// TwinCAT 3 PLC project DynamicDuos
// ProgramVersion: 3.1.4024.0
// libraries:
//   Tc2_Standard, * (Beckhoff Automation GmbH)
//   Tc2_System, * (Beckhoff Automation GmbH)
//   Tc2_Utilities, * (Beckhoff Automation GmbH)
//   Tc3_Module, * (Beckhoff Automation GmbH)
//   Haptix-Beckhoff,newest,HaptiX Lab
// project tree:
//   DUTs/ ActiveWindowStateType.TcDUT, CalibStateType.TcDUT, MainStateType.TcDUT, MasterStateType.TcDUT, ST_CalibLogChunk.TcDUT, ST_CalibrationSettings.TcDUT, ST_CalibTrialStep.TcDUT, ST_LoadExperimentSetting.TcDUT, ST_MainTrialStep.TcDUT
//   GVLs/ GVL.TcGVL
//   / PlcTask.TcTTO
//   POUs/ CalibrationBlock.TcPOU, CalibrationBlockLogger.TcPOU, CalibrationBlock_DOCILE.TcPOU, MAIN.TcPOU, MainExperimentBlock.TcPOU, MainExperimentBlockLogger.TcPOU, MAIN_DOCILE.TcPOU, TEST.TcPOU, WaitingMonitorBlock.TcPOU, MetadataBlock.TcPOU, MotorTorqueToCommandV.TcPOU
// real-time tasks:
//   TASK PlcTask: cycle T#100us, priority 4, ADS port 350
// I/O:
//   DEVICE Device 2 (EtherCAT), AmsNetId 141.212.76.55.3.1
//     Term 1 (EK1100) [EK1100 EtherCAT Coupler (2A E-Bus)]
//       Term 2 (EL4038) [EL4038 8Ch. Ana. Output +/-10V, 12bit]
//       Term 3 (EL3174) [EL3174 4Ch. Ana. Input +/-10V Diff., +/-20mA SingleEnded, 16 Bit]
//       Term 4 (EL5122) [EL5122 2Ch. Inc. Encoder 5V (2xAB TTL)]
//       Term 5 (EL9011) [EL9011 End Terminal]
// variable links:
//   DynamicDuos/DynamicDuos Instance <-> Device 2 (EtherCAT)/Term 1 (EK1100)/Term 2 (EL4038)
//     PlcTask Outputs/MAIN_DOCILE.fbMotor1.nNegAnalogOutput <-> AO Outputs Channel 2/Analog output
//     PlcTask Outputs/MAIN_DOCILE.fbMotor1.nPosAnalogOutput <-> AO Outputs Channel 1/Analog output
//     PlcTask Outputs/MAIN_DOCILE.fbMotor1.nZeroRefAnalogOutput <-> AO Outputs Channel 3/Analog output
//   DynamicDuos/DynamicDuos Instance <-> Device 2 (EtherCAT)/Term 1 (EK1100)/Term 3 (EL3174)
//     PlcTask Inputs/MAIN_DOCILE.fbLoadCell.nAnalogReading <-> AI Standard Channel 1/Value
//   DynamicDuos/DynamicDuos Instance <-> Device 2 (EtherCAT)/Term 1 (EK1100)/Term 4 (EL5122)
//     PlcTask Inputs/GVL.ENCODER_1_A_STATUS <-> ENC Status Channel 1/Status of input A
//     PlcTask Inputs/GVL.ENCODER_1_B_STATUS <-> ENC Status Channel 1/Status of input B
//     PlcTask Inputs/MAIN_DOCILE.fbEncoder1.QE_CHANNEL_COUNTS <-> ENC Status Channel 1/Counter value

CONFIGURATION DynamicDuos
    RESOURCE PLC ON TwinCAT3
        TASK PlcTask(INTERVAL := T#100us, PRIORITY := 4);
        PROGRAM MAIN_DOCILE WITH PlcTask : MAIN_DOCILE;
    END_RESOURCE
END_CONFIGURATION

// ---- DUTs/ActiveWindowStateType.TcDUT
{attribute 'qualified_only'}
{attribute 'strict'}
TYPE ActiveWindowStateType :
(
	EXPERIMENT_WINDOW := 0,
	CALIBRATION_WINDOW := 1, 
	PARTICIPANT_WINDOW := 2, 
	TRACKING_WINDOW := 3
) SINT := EXPERIMENT_WINDOW;
END_TYPE

// ---- DUTs/CalibStateType.TcDUT
{attribute 'qualified_only'}
{attribute 'strict'}
TYPE CalibStateType :
(
	PRE_LAUNCH := 0, // When the user is inputting settings. 
	TEST_SETUP := 1, // When the automation is getting the test ready
	TEST_ACTIVE := 2, // When the test is actively running. 
	TEST_FINISHED := 3, // When all calibration rounds have been completed. 
	ABORT := -1 // When the user has interrupted a test. 
	
);
END_TYPE

// ---- DUTs/MainStateType.TcDUT
{attribute 'qualified_only'}
{attribute 'strict'}
{attribute 'to_string'}
TYPE MainStateType :
(
	PRE_LAUNCH := 0, // When the user is inputting settings. 
	TEST_SETUP := 1, // When the automation is getting the test ready
	TEST_ACTIVE := 2, // When the test is actively running. 
	TEST_FINISHED := 3, // When all calibration rounds have been completed. 
	PROCESSING_LOG := 4, // When the log is saving.
	WAITING_FOR_RELEASE := 5, 
	ABORT := -1 // When the user has interrupted a test. 
);
END_TYPE

// ---- DUTs/MasterStateType.TcDUT
{attribute 'qualified_only'}
{attribute 'strict'}
{attribute 'to_string'}
TYPE MasterStateType :
(
	WAITING := 0, 
	CALIBRATION := 1, 
	ACTIVE := 2,
	TRACKING := 3, 
	ERROR := -1
)SINT := WAITING;
END_TYPE

// ---- DUTs/ST_CalibLogChunk.TcDUT
TYPE ST_CalibLogChunk :
STRUCT
	nChunkSizeBytes : DINT; 
	nChunkIndex : DINT; 
	nLastPointIndex : DINT := -1; // This will be positive if the last data point in an entire log lies within this chunk. The index will be the index of the last data point. 
	aChunk : ARRAY[0..GVL.MAX_CHUNK_SIZE] OF ST_CalibTrialStep;
END_STRUCT
END_TYPE

// ---- DUTs/ST_CalibrationSettings.TcDUT
TYPE ST_CalibrationSettings :
STRUCT
	bTestTypeHuman : BOOL; 
	nNumTrials : UINT;
	bTogglePulseWithGrip : BOOL;  
	bUseManualPulseTimer : BOOL; 
	bUseConstantGripTrigger : BOOL; 
	bUseConstantPulseTorque : BOOL; 
	rConstantPulseTorqueVal : REAL; 
	aGripSchedule : ARRAY[1..100] OF REAL; // There is never going to be 100, just some upper bound.
END_STRUCT
END_TYPE

// ---- DUTs/ST_CalibTrialStep.TcDUT
TYPE ST_CalibTrialStep : // Defines the configuration and data for a calibration trial at a given point in time. 
STRUCT
	nTimestepLow : UDINT;
	nTimeStepHigh : UDINT; 
	rEncoderDegrees : REAL; 
	rEncoderRadians : REAL; 
	rCommandVoltage : REAL; 
	rCommandTorque : REAL; 
	rAppliedTorque : REAL; 
	rVirtualSpringTorque : REAL; 
	rGripForce : REAL; 
	rCurrentGripThreshold : REAL; 
	sSequenceStateString : T_MaxString;  // String of the state
	nCurrentTestIndex : INT;
	nTestIsLive : INT; 
END_STRUCT
END_TYPE

// ---- DUTs/ST_LoadExperimentSetting.TcDUT
TYPE ST_LoadExperimentSetting :
STRUCT
	Weight : INT; 
	Test_Finished : BOOL; 
END_STRUCT
END_TYPE

// ---- DUTs/ST_MainTrialStep.TcDUT
TYPE ST_MainTrialStep :
STRUCT
	nTimestepLow : UDINT; 
	nTimestepHigh : UDINT; 
	rEncoderDegrees : REAL; 
	rEncoderRadians : REAL; 
	rCommandVoltage : REAL; 
	rCommandTorque : REAL; 
	rWallTorque : REAL; 
	rGripForce : REAL; 
	sSequenceStateString : T_MaxString; 
	nCurrentTestIndex : INT; 
	nTestIsLive : INT; 
END_STRUCT
END_TYPE

// ---- GVLs/GVL.TcGVL
{attribute 'qualified_only'}
VAR_GLOBAL

	ENCODER_1_DEGREES : REAL; 
	ENCODER_1_COUNTER_VALUE : LINT; 
	MOTOR_1_APPLIED_VOLTAGE : REAL; 
	ENCODER_1_A_STATUS AT %I* : BOOL; 
	ENCODER_1_B_STATUS AT %I* : BOOL;
	LOAD_CELL_NEWTONS : REAL; 
	MAIN_SYSTEM_TIME : UDINT; 
	CALIB_SYSTEM_TIME : UDINT; 
	
END_VAR

VAR_GLOBAL CONSTANT
	// Max amount of data entries we can 
	// send over the wire at once. 
	MAX_CHUNK_SIZE : DINT := 100; 
END_VAR

// ---- POUs/MAIN_DOCILE.TcPOU
PROGRAM MAIN_DOCILE
VAR
	
	// Variables for logging
	nEncoderCounts : LINT; 
	rEncoderDegrees : REAL;
	rEncoderLastDegrees : REAL; 
	rEncoderRadians : REAL; 
	rEncoderLastRadians : REAL; 
	rEncoderRadiansBuffer : ARRAY[1..FILTER_WINDOW] OF REAL; 
	rEncoderRadiansSum : REAL; 
	rEncoderRadiansFiltered : REAL; 
	nFilterBufferCount : INT := 0; 
	rGripForce : REAL; 
	
	// Sensors instantiation 
	fbEncoder1 : FB_QuadratureEncoder;
	fbLoadCell : FB_AnalogLoadCellInput;
	fbMotor1 : FB_AnalogMotorDriver;	

	
	// Helpers
	i : INT := 0;
	j : INT := 0;
	bIsFirstReset : BOOL := TRUE; 
	bEncoderReset : BOOL := FALSE; 
	fbSystemTime : GETSYSTEMTIME;
	
	stMasterState : MasterStateType := MasterStateType.WAITING; 
	
	
	// Child function block 
	{attribute 'OPC.UA.DA':='1'}
	fbCalibrationBlock : CalibrationBlock_DOCILE; 
	
	testCalibrationSettings : ST_CalibrationSettings; 

END_VAR
VAR CONSTANT
	// Constants for digital filtering 
	FILTER_WINDOW : INT := 11; 
END_VAR

// ===================================================== COMPLETE ALL SENSOR READINGS ========================================================
IF bIsFirstReset OR bEncoderReset THEN 
	fbEncoder1.Reset();
	bIsFirstReset := FALSE;
	bEncoderReset := FALSE; 
END_IF

// Encoders 
fbEncoder1(); 
nEncoderCounts := fbEncoder1.nNetCounts; 
rEncoderDegrees := fbEncoder1.rDegrees; 
rEncoderLastDegrees := fbEncoder1.rLastDegrees; 
rEncoderRadians := fbEncoder1.rRadians; 
rEncoderLastRadians := fbEncoder1.rLastRadians;

// Update digital filter. 
IF nFilterBufferCount < FILTER_WINDOW THEN 
	nFilterBufferCount := nFilterBufferCount + 1; 
END_IF

// Shift the buffer and add the new reading 
FOR i := FILTER_WINDOW TO 2 BY -1 DO
	rEncoderRadiansBuffer[i] := rEncoderRadiansBuffer[i-1]; 
END_FOR
rEncoderRadiansBuffer[1] := rEncoderRadians;

// Compute the moving average only if the buffer is full
j := MIN(nFilterBufferCount, FILTER_WINDOW); 
rEncoderRadiansSum := 0.0; 
FOR i:= 1 TO j DO
	rEncoderRadiansSum := rEncoderRadiansSum + rEncoderRadiansBuffer[i];
END_FOR
rEncoderRadiansFiltered := rEncoderRadiansSum / j; 

// Load cell   
fbLoadCell(); 
rGripForce := fbLoadCell.rCalibratedOutput; 
// ================================================ END SENSOR READINGS ==================================================

IF stMasterState = MasterStateType.CALIBRATION THEN 
	fbCalibrationBlock(
		rEncoderRadians := rEncoderRadians,
		rEncoderRadiansFiltered := rEncoderRadiansFiltered,
		rEncoderLastRadians := rEncoderLastRadians, 
		rGripForce := rGripForce,
		fbMotorReference := fbMotor1
	);
END_IF



// ================================================= UPDATE THE GVL ======================================================
GVL.ENCODER_1_DEGREES := fbEncoder1.rDegrees; 
GVL.LOAD_CELL_NEWTONS := rGripForce; 
fbSystemTime(timeLoDW => GVL.MAIN_SYSTEM_TIME);

END_PROGRAM

// ---- POUs/CalibrationBlock_DOCILE.TcPOU
FUNCTION_BLOCK CalibrationBlock_DOCILE
VAR_INPUT
	rEncoderRadians : REAL ;
	rEncoderRadiansFiltered : REAL; 
	rEncoderLastRadians : REAL;
	rGripForce : REAL; 
	fbMotorReference : REFERENCE TO FB_AnalogMotorDriver; 
END_VAR
VAR_OUTPUT
	rCommandVoltage : REAL;
	rVirtualSpringTorque : REAL;
	rAppliedTorque : REAL; 
	rCommandTorque : REAL; 
	rError : REAL;
	rLastError : REAL := 0;
	rProportional : REAL;
	rIntegral : REAL := 0;
	rDerivative : REAL; 
	bPIDStale : BOOL := TRUE; 
	rControlOutput : REAL;
	Kp : REAL := 0.3;
	Ki : REAL := 0.03;
	Kd : REAL := 0.05; 
	d_time : REAL := 0.0001; 
END_VAR
VAR
	z : INT := 0; 
	
	// State machine members for executing the test
	eSequenceState : CalibStateType := CalibStateType.PRE_LAUNCH; 
	eNextSequenceState : CalibStateType := CalibStateType.PRE_LAUNCH; 
	eSetupSubState : (HOMING, WAITING); 
	stCalibStepState : ST_CalibTrialStep; 
	stCalibrationSettings : ST_CalibrationSettings;
	
	// Virtual timers for accessing the test
	fbTonTest : TON := (PT := T#1000MS); // Timer for the entire test
	fbTonPulse : TON := (PT := T#200MS); // Timer for the duration of the pulse
	fbTonHoming : TON := (PT := T#500MS); // Time to give state machine to home
	bMotorLimitHit : BOOL := FALSE; 
	bWheelIsIdle : BOOL; 
	bTestIsLive : BOOL := FALSE; 
	bTestIsLiveTrigger : BOOL := FALSE; 
	rStartGripThreshold : REAL := 1.5;
	nCurrentTestIndex : INT := 0; 
	bLaunchTestSequence: BOOL;
	rCurrentGripThreshold : REAL := 100; // High number for init just so it can't go off by itself
	nCurrentLaunchIndex: INT := 0; 
	bLogHasBeenAcknowledged : BOOL := FALSE; 
	
	// Helper functions
	fbSystemTime : GETSYSTEMTIME; 
	nLastTimeStep : UDINT; 
	fbLogger : CalibrationBlockLogger; 
END_VAR

// Update the timers
fbTonTest(IN := bTestIsLive); 
fbTonPulse(IN := bTestIsLive);

CASE eSequenceState OF 
	
	// The user is currently setting prelaunch settings. 
	CalibStateType.PRE_LAUNCH: 
	
		// Make sure all variables are zerod 
		bTestIsLive := FALSE;
		rCommandVoltage := 0; 
		rVirtualSpringTorque := 0; 
		rAppliedTorque := 0; 
		rCommandTorque := 0; 
		fbMotorReference(rCommandVoltage := rCommandVoltage); 
	
		IF bLaunchTestSequence THEN // This would be set by the "LaunchTestSequence" method.
			eNextSequenceState := CalibStateType.TEST_SETUP; 
			
			// Also set the first test index
			nCurrentTestIndex := 1;  
			bLaunchTestSequence := FALSE; 
		ELSE
			eNextSequenceState := CalibStateType.PRE_LAUNCH; 
		END_IF
		
	// We are getting the test readt 
	CalibStateType.TEST_SETUP: 
	
		CASE eSetupSubState OF 
			HOMING: 
			
				bMotorLimitHit := FALSE; 
				
				// In this state, we need to recenter the motor back to the 0 point 
				// afterwards, we need to wait for the trigger signal 
				rError := 0 - rEncoderRadiansFiltered; 
				rProportional := Kp * rError; 
				rIntegral := rIntegral + (rError * d_time); 
				rDerivative := (rError - rLastError) / d_time; 
				rLastError := rError; 
				
				// On the first step, if the PID is stale, just use proportional 
				IF bPIDStale THEN 
					rAppliedTorque := rProportional; 
					rIntegral := 0; 
					bPIDStale := FALSE; 
				ELSE
					rAppliedTorque := rProportional + (Ki * rIntegral) + (Kd * rDerivative); 
				END_IF
				rVirtualSpringTorque := 0; 
				rCommandTorque := rAppliedTorque + rVirtualSpringTorque; 
				rCommandVoltage := MotorTorqueToCommandV(rCommandTorque := rCommandTorque); 
				fbMotorReference(rCommandVoltage := rCommandVoltage); 
				
				// Check to see if the wheel has been idle for ong enough 
				bWheelIsIdle := rGripForce < rStartGripThreshold AND ABS(rEncoderRadians) < 0.08;
				fbTonHoming(IN := bWheelIsIdle); 
				
				IF fbTonHoming.Q THEN 
					eSetupSubState := WAITING; 
				END_IF
				
			WAITING: 
				
				// Then we need to check if the test launch conditions are met 
				// We need to figure out the type of trigger being used
				IF bTestIsLiveTrigger AND NOT stCalibrationSettings.bTogglePulseWithGrip THEN
					bTestIsLive := TRUE; 
					bTestIsLiveTrigger := FALSE; 
				END_IF
				
				// If it's not the above, then we are toggling pulse with grip 
				IF  stCalibrationSettings.bTogglePulseWithGrip THEN 
					IF stCalibrationSettings.bUseConstantGripTrigger THEN 
						rCurrentGripThreshold := stCalibrationSettings.aGripSchedule[1]; 
					ELSE
						rCurrentGripThreshold := stCalibrationSettings.aGripSchedule[nCurrentTestIndex];
					END_IF 
					
					// Once we've set the value, we can compare to see if we've reached it
					IF rGripForce > rCurrentGripThreshold THEN 
						bTestIsLive := TRUE; 
					END_IF
					
				END_IF
				
				IF bTestIsLive THEN 
					eNextSequenceState := CalibStateType.TEST_ACTIVE; 
					bWheelIsIdle := FALSE; 
					fbTonHoming(IN := bWheelIsIdle); 
					eSetupSubState := HOMING; 
					bPIDStale := TRUE; 
				ELSE
					eNextSequenceState := CalibStateType.TEST_SETUP;
					// We need to let go of the motor
					rVirtualSpringTorque := 0; 
					rAppliedTorque := 0; 
					rCommandTorque := 0; 
					rCommandVoltage := 0;
					fbMotorReference(rCommandVoltage := rCommandVoltage); 
				END_IF
				
				
		END_CASE
		
		
	/// Then we handle the logic for actually completing the test 
	CalibStateType.TEST_ACTIVE: 
	
			// Timer is set based on the bTestIsLive variable. 
			IF NOT fbTonPulse.Q THEN 
			
				// We want to split motor action between motor test and human test mode. 
				// In motor test mode, we add a virtual spring so the motor doesn't slam into the bale
				IF NOT stCalibrationSettings.bTestTypeHuman THEN
					
					rAppliedTorque := stCalibrationSettings.rConstantPulseTorqueVal; 
					rVirtualSpringTorque := -1 * 0.35 * rEncoderRadians; 
				ELSE
					
					IF NOT stCalibrationSettings.bUseConstantPulseTorque THEN 
						rAppliedTorque := 0.4 + 0.02 * rCurrentGripThreshold; 
					ELSE
						rAppliedTorque := stCalibrationSettings.rConstantPulseTorqueVal; 
					END_IF 
					rVirtualSpringTorque := 0; 
			
				END_IF
				
				rCommandTorque := rAppliedTorque + rVirtualSpringTorque; 
				rCommandVoltage := MotorTorqueToCommandV(rCommandTorque := rCommandTorque); 
			ELSE
				
				IF NOT stCalibrationSettings.bTestTypeHuman THEN 
					rAppliedTorque := 0; 
					rVirtualSpringTorque := -1 * 0.35 * rEncoderRadians; 
				ELSE
					rAppliedTorque := 0; 
					rVirtualSpringTorque := 0; 
				END_IF
				
				rCommandTorque := rAppliedTorque + rVirtualSpringTorque; 
				rCommandVoltage := MotorTorqueToCommandV(rCommandTorque := rCommandTorque); 
			END_IF
			
			fbMotorReference(rCommandVoltage := rCommandVoltage); 
			
			// Now we check the test timer
			IF fbTonTest.Q THEN
				bTestIsLive := FALSE;
				IF nCurrentTestIndex < UINT_TO_INT(stCalibrationSettings.nNumTrials) THEN 
					nCurrentTestIndex := nCurrentTestIndex + 1; 
					eNextSequenceState := CalibStateType.TEST_SETUP; 
				ELSE
					eNextSequenceState := CalibStateType.TEST_FINISHED;
				END_IF
			END_IF
	
	CalibStateType.TEST_FINISHED: 
		// Do some logging 
		IF NOT bLogHasBeenAcknowledged THEN 
			eNextSequenceState := CalibStateType.TEST_FINISHED; 
		END_IF
		eNextSequenceState := CalibStateType.PROCESSING_LOG;
		
	CalibStateType.PROCESSING_LOG: 
		// Wait to see if logging finished
		nCurrentTestIndex := 0; 
		nCurrentLaunchIndex := nCurrentLaunchIndex + 1; 
		eNextSequenceState := CalibStateType.PRE_LAUNCH; 
END_CASE


// At the end of the main loop is when we actually do the logging 
nLastTimeStep := stCalibStepState.nTimestepLow; 
fbSystemTime(timeLoDW => stCalibStepState.nTimestepLow, timeHiDW => stCalibStepState.nTimeStepHigh); 
stCalibStepState.rEncoderDegrees := RAD_TO_DEG(rEncoderRadians); 
stCalibStepState.rEncoderRadians := rEncoderRadians; 
stCalibStepState.rCommandVoltage := rCommandVoltage; 
stCalibStepState.rCommandTorque := rCommandTorque; 
stCalibStepState.rAppliedTorque := rAppliedTorque; 
stCalibStepState.rVirtualSpringTorque := rVirtualSpringTorque; 
stCalibStepState.rGripForce := rGripForce; 
stCalibStepState.rCurrentGripThreshold := rCurrentGripThreshold; 
stCalibStepState.sSequenceStateString := TO_STRING(eSequenceState); 
stCalibStepState.nCurrentTestIndex := nCurrentTestIndex; 
stCalibStepState.nTestIsLive := BOOL_TO_INT(bTestIsLive); 

IF eSequenceState = CalibStateType.TEST_ACTIVE THEN
	fbLogger.addStep(stNewStep := stCalibStepState);
END_IF

// Update sequence state for next iteration 
eSequenceState := eNextSequenceState;

END_FUNCTION_BLOCK

// ---- POUs/CalibrationBlockLogger.TcPOU
FUNCTION_BLOCK CalibrationBlockLogger
VAR_INPUT
	sFileName : STRING; 
END_VAR
VAR_OUTPUT
	bBusy : BOOL := FALSE; 
	bError : BOOL := FALSE; 
END_VAR
VAR CONSTANT
	nMaxBufferSize : UDINT := 2000000;
END_VAR
VAR
	cDefaultHeader : T_MaxString := 'TimeLow,TimeHigh,EncoderDegrees,EncoderRadians,CommandVoltage,CommandTorque,AppliedTorque,VSTorque,GripForce,GripThreshold,SequenceState,CurrentTestIndex,TestIsLive $n'; 
	sDefaultDirectory : T_MaxString := 'C:\Users\njanne\Documents\DDTestLogs\calibration\'; 
	bWriteToDisk : BOOL := FALSE; 
	eFileWriteState : (IDLE, OPEN, WRITE, CLOSE, ERROR); 
	nFileWriteSubstep : INT := 0; 
	fbFileOpen : FB_FileOpen; 
	fbFilePuts : FB_FilePuts; 
	fbFileClose : FB_FileClose; 
	fbFormatString : FB_FormatString2; 
	nFileHandle : UINT; 
	bHeaderWriteComplete : BOOL := FALSE; 
	nWriteIndex : UDINT := 0; 
	sWritePercentFormat : T_MaxString := '%.2f %%'; 
	rWritePercent : REAL; 
	sWritePercentString : T_MaxString; 
	
	// For formatting data into a string. 
	sDataFormatStr1 : STRING := '%d,%d,%f,%f,%f,%f,%f,'; 
	sDataFormatStr2 : STRING := '%f,%f,%f,%s,%d,%d $n';
	sTempString : STRING(600); 
	sOutputString : STRING(600); 
	
	aTrialDataBuffer : ARRAY[0..nMaxBufferSize] OF ST_CalibTrialStep; 
	nStepsSoFar : UDINT := 0; // Current number of steps in the database. 
	
END_VAR

IF bWriteToDisk THEN

	// If it's time to write to disk, we need to empty the buffer.
	CASE eFileWriteState OF 
		
		IDLE: 
			// Get everything ready. 
			nFileHandle := 0; 
			bBusy := TRUE; 
			eFileWriteState := OPEN;
			nFileWriteSubstep := 0;  
	
		OPEN:
			CASE nFileWriteSubstep OF
				0:  
					// Opens a file for writing at the end of the file (append). 
					// If the file does not exist, a new file is created. 
					fbFileOpen(spathName := CONCAT(sDefaultDirectory, sFilename), bExecute := FALSE); 
					fbFileOpen(
						bExecute 		:= TRUE, 
						sNetID			:= '',
						sPathName 		:= CONCAT(sDefaultDirectory, sFilename), 
						nMode 			:= FOPEN_MODEAPPEND OR FOPEN_MODETEXT); 
		
					nFileWriteSubstep := nFileWriteSubstep + 1; // Advance to waiting state. 
	
				1: 
					fbFileOpen(bExecute := FALSE); 
					IF NOT fbFileOpen.bBusy THEN 
						IF fbFileOpen.bError THEN 
							eFileWriteState := ERROR; 
							nFileWriteSubstep := 0; 
						ELSE
							nFileHandle := fbFileOpen.hFile; 
							eFileWriteState := WRITE; 
							nFileWriteSubstep := 0; 
						END_IF
					END_IF
				END_CASE

		WRITE: 
			CASE nFileWriteSubstep OF 
				0 :
					fbFilePuts(bExecute := FALSE); 
					
					// Check if we still need to write the header. 
					IF NOT bHeaderWriteComplete THEN
						fbFilePuts(
							bExecute		:= TRUE, 
							sNetId			:= '', 
							hFile			:= nFileHandle, 
							sLine			:= cDefaultHeader);
						bHeaderWriteComplete := TRUE; 
					ELSE
						// If the header is already written, then we're going for data. 
						// We need to first format the string. 		
						fbFormatString(
							pFormatString := ADR(sDataFormatStr1), 
							arg1 := F_UDINT(aTrialDataBuffer[nWriteIndex].nTimestepLow), 
							arg2 := F_UDINT(aTrialDataBuffer[nWriteIndex].nTimeStepHigh),
							arg3 := F_REAL(aTrialDataBuffer[nWriteIndex].rEncoderDegrees), 
							arg4 := F_REAL(aTrialDataBuffer[nWriteIndex].rEncoderRadians), 
							arg5 := F_REAL(aTrialDataBuffer[nWriteIndex].rCommandVoltage), 
							arg6 := F_REAL(aTrialDataBuffer[nWriteIndex].rCommandTorque), 
							arg7 := F_REAL(aTrialDataBuffer[nWriteIndex].rAppliedTorque), 
							pDstString := ADR(sOutputString), 
							nDstSize := SIZEOF(sOutputString)); 
					
						fbFormatString(
							pFormatString := ADR(sDataFormatStr2), 
							arg1 := F_REAL(aTrialDataBuffer[nWriteIndex].rVirtualSpringTorque), 
							arg2 := F_REAL(aTrialDataBuffer[nWriteIndex].rGripForce), 
							arg3 := F_REAL(aTrialDataBuffer[nWriteIndex].rCurrentGripThreshold), 
							arg4 := F_STRING(aTrialDataBuffer[nWriteIndex].sSequenceStateString), 
							arg5 := F_INT(aTrialDataBuffer[nWriteIndex].nCurrentTestIndex), 
							arg6 := F_INT(aTrialDataBuffer[nWriteIndex].nTestIsLive), 
							pDstString := ADR(sTempString), 
							nDstSize := SIZEOF(sTempString)); 
							
						CONCAT2(
							pSrcString1 := ADR(sOutputString), 
							pSrcString2 := ADR(sTempString), 
							pDstString := ADR(sOutputString), 
							nDstSize := SIZEOF(sOutputString)); 
						
						fbFilePuts(
							bExecute		:= TRUE, 
							sNetId			:= '', 
							hFile			:= nFileHandle, 
							sLine			:= sOutputString); 
							
						nWriteIndex := nWriteIndex + 1; 
						// Update write progress 
						rWritePercent := UDINT_TO_REAL(nWriteIndex) / UDINT_TO_REAL(nStepsSoFar) * 100; 
						fbFormatString(
							pFormatString := ADR(sWritePercentFormat),
							arg1 := F_REAL(rWritePercent),
							pDstString := ADR(sWritePercentString), 
							nDstSize := SIZEOF(sWritePercentString)); 
				
					END_IF
					
					nFileWriteSubstep := nFileWriteSubstep + 1; // Advance to waiting state. 
					
				1 : 
					fbFilePuts(bExecute := FALSE); 
					IF NOT fbFilePuts.bBusy THEN
						IF fbFilePuts.bError THEN 
							eFileWriteState := ERROR; 
							nFileWriteSubstep := 0; 
						ELSE
							// Check if we have more things to write to the CSV still
							IF nWriteIndex = nStepsSoFar THEN
								eFileWriteState := CLOSE; 
							ELSE
								eFileWriteState := WRITE;
							END_IF 
						END_IF
						nFileWriteSubstep := 0; 
					END_IF
					
					
			END_CASE
		
		CLOSE: 
			CASE nFileWriteSubstep OF
				0: 
					fbFileClose(bExecute := FALSE); 
					fbFileClose(
						bExecute	:= TRUE, 
						sNetId		:= '', 
						hFile		:= nFileHandle); 
					nFileWriteSubstep := nFileWriteSubstep + 1; 
					
				1: 
					fbFileClose(bExecute := FALSE); 
					IF NOT fbFileClose.bBusy THEN
						IF fbFileClose.bError THEN 
							eFileWriteState := ERROR; 
							nFileWriteSubstep := 0; 
						ELSE
							eFileWriteState := IDLE; 
							nFileHandle := 0; 
							
							// Also reset everything so that a new test can overrite 
							nStepsSoFar := 0; 
							nWriteIndex := 0; 
							nFileWriteSubstep := 0; 
							bHeaderWriteComplete := FALSE; 
							bBusy := FALSE; 
							bWriteToDisk := FALSE; 
						END_IF
						
					END_IF
			END_CASE
				
		ERROR: 
			// Error, clear the handle and go back to idle. 
			nFileHandle := 0; 
			eFileWriteState := IDLE; 
			bError := TRUE; 
	
	END_CASE

END_IF

METHOD addStep : BOOL
VAR_INPUT
	stNewStep : ST_CalibTrialStep; // The incoming step to be added to memory
END_VAR
// We need to simply copy over all the fields into the new position. 
// And then, update the counter. 
MEMCPY(
	destAddr := ADR(aTrialDataBuffer[nStepsSoFar]), 
	srcAddr := ADR(stNewStep), 
	n := SIZEOF(ST_CalibTrialStep)); 
	
nStepsSoFar := nStepsSoFar + 1;
END_METHOD

{attribute 'TcRpcEnable':='1'}
METHOD getLogChunk : ST_CalibLogChunk
VAR_INPUT
	nChunkIndex : DINT; 
END_VAR
VAR
	nRemainingPts : DINT; 
END_VAR
// We essentially want to copy the indices from 
// chunk index + max_chunk_size into the array that is sitting in the
// return type 
getLogChunk.nChunkIndex := nChunkIndex; 

IF ((nChunkIndex * GVL.MAX_CHUNK_SIZE + GVL.MAX_CHUNK_SIZE) <= nStepsSoFar) THEN
	getLogChunk.nChunkSizeBytes := GVL.MAX_CHUNK_SIZE*SIZEOF(ST_CalibTrialStep);
	MEMCPY(ADR(getLogChunk.aChunk), ADR(aTrialDataBuffer[nChunkIndex*GVL.MAX_CHUNK_SIZE]), getLogChunk.nChunkSizeBytes); 
ELSE
	nRemainingPts := nStepsSoFar - nChunkIndex * GVL.MAX_CHUNK_SIZE; 
	getLogChunk.nChunkSizeBytes := nRemainingPts*SIZEOF(ST_CalibTrialStep);
	MEMCPY(ADR(getLogChunk.aChunk), ADR(aTrialDataBuffer[nChunkIndex*GVL.MAX_CHUNK_SIZE]), getLogChunk.nChunkSizeBytes); 
	getLogChunk.nLastPointIndex := nRemainingPts; 
END_IF
END_METHOD

{attribute 'TcRpcEnable':='1'}
METHOD getLogSize : BOOL
VAR_INPUT
END_VAR
VAR_OUTPUT
	nCurrentChunkSize : DINT := GVL.MAX_CHUNK_SIZE; 
	nNumLogPoints : DINT := nStepsSoFar;
	nNumLogChunks : DINT; 
	nSizeLastChunk : DINT; 
	nLogSizeBytes : DINT := nStepsSoFar * SIZEOF(ST_CalibTrialStep); 
END_VAR
nNumLogChunks := nStepsSoFar / GVL.MAX_CHUNK_SIZE;
nSizeLastChunk := nStepsSoFar MOD GVL.MAX_CHUNK_SIZE; 

IF (nSizeLastChunk <> 0) THEN
	nNumLogChunks := nNumLogChunks + 1; // Since the last chunk is there, just smaller
ELSE
	// If somehow we have exactly as many data points that can be divided evenly into chunks
	nSizeLastChunk := GVL.MAX_CHUNK_SIZE; 
END_IF

// Also return false if there is no log 
IF nStepsSoFar = 0 THEN 
	getLogSize := FALSE;
ELSE
	getLogSize := TRUE; 
END_IF
END_METHOD

METHOD writeLog : BOOL
VAR_INPUT
END_VAR
bWriteToDisk := TRUE;
END_METHOD

END_FUNCTION_BLOCK

// ---- POUs/MotorTorqueToCommandV.TcPOU
FUNCTION MotorTorqueToCommandV : REAL // Calculates the voltage to send to the motor given a requested torque
// NOTE: Needs to be calibrated from time to time. 
VAR_INPUT
	rCommandTorque : REAL; // N-m
END_VAR
VAR
	// Equation is of the form rCommandVoltage = rVoltageSlope*(rCommandTorque) + rVoltageIntercept
	// Exact values are found from calibration. 
	rVoltageSlope : REAL := 9.26; 
	rVoltageIntercept : REAL := 0.0758; 
END_VAR

MotorTorqueToCommandV := rVoltageSlope * rCommandTorque + rVoltageIntercept;

END_FUNCTION

// ---- POUs/CalibrationBlock.TcPOU
FUNCTION_BLOCK CalibrationBlock
VAR_INPUT

	fbMotorReference : REFERENCE TO FB_AnalogMotorDriver; 
	fbMetadata : REFERENCE TO MetadataBlock; 	

END_VAR
VAR_OUTPUT

	// Variables for logging 
	nEncoderCounts : LINT; 
	rEncoderDegrees : REAL; 
	rEncoderLastDegrees : REAL; 	
	rEncoderRadians : REAL; 
	rEncoderLastRadians : REAL; 
	rEncoderRadiansBuffer : ARRAY[1..FILTER_WINDOW] OF REAL; 
	rEncoderRadiansSum : REAL; 
	rEncoderRadiansFiltered : REAL; 
	nFilterBufferCount : INT := 0; 
	
	// Variables for motor control 
	rCommandVoltage : REAL; 
	rVirtualSpringTorque : REAL; // Torque applied by any vritual spring
	rAppliedTorque : REAL;  // Torque applied as part of the test
	rCommandTorque : REAL; // The sum of the two variables above.  
		rError : REAL; 
	rLastError : REAL; 
	rProportional : REAL; 
	rIntegral : REAL := 0; 
	rDerivative : REAL; 
	bPIDStale : BOOL := TRUE;
	rControlOutput : REAL; 
	Kp : REAL := 0.3; 
	Ki : REAL := 0.03; 
	Kd : REAL := 0.05; 
	d_time : REAL := 0.0001; // Time step (100 us). 
	
	// Variables for load cell 
	rGripForce : REAL; 

END_VAR

// Constants used for the program 
VAR CONSTANT
	rAngleNormalizationFactor : REAL := 90; 
	nMaxTrialNumber : UINT := 10; 
	FILTER_WINDOW : INT := 11; 
END_VAR

VAR
	
	// Variables to keep track of the actual encoder/motor setup
	fbEncoder1 : FB_QuadratureEncoder; 
	fbLoadCell : FB_AnalogLoadCellInput; // TODO: Change everything to top level reference maybe? 
	
	////// BEGIN GUI TEST OPTIONS
	//// All fields in the next section are in some way or another set by the GUI, and define 
	//// the type of test to take place.
	// 1. Test type
	bTestTypeHuman : BOOL; // Whether or not this a human or motor test 
	bTestTypeHumanLIVE : BOOL; 
	
	// 2. Number of trials
	nTrialNumber : UINT := 1; // Number of calibration trials to run in succession 
	nTrialNumberLIVE : UINT; 
	
	// 3. Trigger type
	bManualPulse : BOOL; // Whether to use manual pulse or grip schedule. 
	bManualPulseLIVE : BOOL; 
	bManualPulseTimerEnable : BOOL; 
	bManualPulseTimerEnableLIVE : BOOL;
	rManualPulseTimerValue : REAL; 
	rManualPulseTimerValueLIVE : REAL;
	
	// 4. Trigger controls
	bUseConstantGripTrigger : BOOL;
	bUseConstantGripTriggerLIVE : BOOL;
	aGripSchedule : ARRAY[1..nMaxTrialNumber] OF REAL;
	aGripScheduleLIVE : ARRAY[1..nMaxTrialNumber] OF REAL;  
	rCurrentGripThreshold : REAL := 0; 
	
	// 5. Pulse controls 
	bUseConstantPulseTorque : BOOL; 
	bUseConstantPulseTorqueLIVE : BOOL;
	rConstantTorqueSetting : REAL; 	
	rConstantTorqueSettingLIVE : REAL;

	// 6. Test Controls
	bLaunchTestSequence : BOOL := FALSE; // Triggers an entry into the testing loop. 
 
	/////// END GUI TEST OPTIONS
	
	// State machine for actual calibration logic. 
	// At the begginning, we are in the configuration state. 
	eSequenceState : CalibStateType := CalibStateType.PRE_LAUNCH; 
	eNextSequenceState : CalibStateType := CalibStateType.PRE_LAUNCH; 
	eSetupSubState : (HOMING, WAITING); 
	nCurrentTestIndex : INT := 0; 
	bTestIsLive : BOOL := FALSE; 
	bTestIsLiveTrigger : BOOL := FALSE; 
	
	// Helper variables 
	i : INT;
	j : INT;  
	fbTonTest : TON := (PT := T#1000MS); // Timer for the entire test
	fbTonPulse : TON := (PT := T#200MS); // Timer for the duration of the pulse 
	fbTonHoming : TON := (PT := T#500MS); // Time to give state machine to home
	bMotorLimitHit : BOOL := FALSE; 
	stCalibStepState : ST_CalibTrialStep; 
	nCurrentLaunchIndex : INT := 0;
	TempString : T_MaxString;
	
	// Helper Functions 
	fbLogger : CalibrationBlockLogger; 
	fbSystemTime : GETSYSTEMTIME; 
	fbFormatString : FB_FormatString; 
	nLastTimeStep : UDINT; 

	bWheelIsIdle: BOOL;
	rStartGripThreshold: REAL := 1.5;
END_VAR

///////////// Read sensors on current iteration
// Encoders 
fbEncoder1(); 
nEncoderCounts := fbEncoder1.nNetCounts; 
rEncoderDegrees := fbEncoder1.rDegrees; 
rEncoderLastDegrees := fbEncoder1.rLastDegrees; 
rEncoderRadians := fbEncoder1.rRadians; 
rEncoderLastRadians := fbEncoder1.rLastRadians; 

// Update digital filter. 
IF nFilterBufferCount < FILTER_WINDOW THEN 
	nFilterBufferCount := nFilterBufferCount + 1; 
END_IF

// Shift the buffer and add the new reading 
FOR i := FILTER_WINDOW TO 2 BY -1 DO
	rEncoderRadiansBuffer[i] := rEncoderRadiansBuffer[i-1]; 
END_FOR
rEncoderRadiansBuffer[1] := rEncoderRadians;

// Computer the moving average only if the buffer is full
j := MIN(nFilterBufferCount, FILTER_WINDOW); 
rEncoderRadiansSum := 0.0; 
FOR i:= 1 TO j DO
	rEncoderRadiansSum := rEncoderRadiansSum + rEncoderRadiansBuffer[i];
END_FOR
rEncoderRadiansFiltered := rEncoderRadiansSum / j; 

// Load cell 
fbLoadCell(); 
rGripForce := fbLoadCell.rCalibratedOutput; 
///////////// End sensor reading 

// Update Timers 
// First we compute the timer update 
fbTonTest(IN := bTestIsLive); 
fbTonPulse(IN := bTestIsLive); 

// Update file object 
// Here we also create the beginning of the logging file. 
// Generate the file name 
fbFormatString(
	sFormat := '%s_test_%d.csv', 
	arg1 := F_STRING(fbMetadata.sUserID), 
	arg2 := F_INT(nCurrentLaunchIndex));
	
fbLogger(sFileName := fbFormatString.sOut); 

// Now we go through the calibration logic. 
CASE eSequenceState OF
	
	// The user is currently setting permissions, we can update them live. 
	CalibStateType.PRE_LAUNCH:
	
		// First we start by updating options to the LIVE variables. 
		bTestTypeHumanLIVE := bTestTypeHuman; 
		nTrialNumberLIVE := nTrialNumber; 
		bManualPulseLIVE := bManualPulse; 
		bManualPulseTimerEnableLIVE := bManualPulseTimerEnable; 
		rManualPulseTimerValueLIVE := rManualPulseTimerValue;
		bUseConstantGripTriggerLIVE := bUseConstantGripTrigger; 
		
		FOR i := 1 TO nMaxTrialNumber DO
			aGripScheduleLIVE[i] := aGripSchedule[i]; 
		END_FOR
		
		bUseConstantPulseTorqueLIVE := bUseConstantPulseTorque;
		rConstantTorqueSettingLIVE := rConstantTorqueSetting; 
		
		IF bLaunchTestSequence THEN
			eNextSequenceState := CalibStateType.TEST_SETUP; 
			// Also set the first test index 
			nCurrentTestIndex := 1; 
			// And put this signal back down 
			bLaunchTestSequence := FALSE; 
				
		ELSE
			eNextSequenceState := CalibStateType.PRE_LAUNCH; 
		END_IF
		
		// We also need to make sure any motor commands are no longer hanging over 
		bTestIsLive := FALSE; 
		rCommandVoltage := 0; 
		rVirtualSpringTorque := 0; 
		rAppliedTorque := 0; 
		rCommandTorque := 0; 
		fbMotorReference(rCommandVoltage := rCommandVoltage); 
		
	// We are getting the test ready. 
	CalibStateType.TEST_SETUP: 
	
		CASE eSetupSubState OF
			HOMING: 
			
				bMotorLimitHit := FALSE; 
				
				// In this state, we need to recenter the motor back to the 0 point, and 
				// we also need to wait for the triggering signal. 
				rError := 0 - rEncoderRadiansFiltered; 
				rProportional := Kp * rError; 
				rIntegral := rIntegral + (rError * d_time); 
				rDerivative := (rError - rLastError) / d_time; 
				rLastError := rError; 
				//rCommandTorque := -1 * ((3/2) * rEncoderRadians - (2/3) * rEncoderLastRadians);
				IF bPIDStale THEN
					rAppliedTorque := rProportional;
					rIntegral := 0; 
					bPIDStale := FALSE; 
				ELSE 
					rAppliedTorque := rProportional + (Ki * rIntegral) + (Kd * rDerivative);
				END_IF
				rVirtualSpringTorque := 0; 
				rCommandTorque := rAppliedTorque + rVirtualSpringTorque; 
				rCommandVoltage := MotorTorqueToCommandV(rCommandTorque := rCommandTorque); 
				fbMotorReference(rCommandVoltage := rCommandVoltage); 
				
				// Check to see if the wheel has been idle for long enough. 
				bWheelIsIdle := rGripForce < rStartGripThreshold AND ABS(rEncoderDegrees) < 5;  
				fbTonHoming(IN := bWheelIsIdle); 
				
				IF fbTonHoming.Q THEN
					eSetupSubState := WAITING; 
				END_IF
				
			WAITING: 
			
				// Then we check to see if the test going live conditions are met: 
				// We need to figure out the type of trigger that's being used, and then we test for that. 
				// In the first scenario, it's if there is a manual pulse sent from the button
				IF bTestIsLiveTrigger AND bManualPulseLIVE AND NOT bManualPulseTimerEnableLIVE THEN // Manually push button 
					bTestIsLive := TRUE; 
					bTestIsLiveTrigger := FALSE; 
				END_IF 
				
				// Then we need to check if it's a grip trigger pulse. To do this, we first update what the grip trigger
				// should be, and then we check to see if the current grip matches that value 
				IF NOT bManualPulseLIVE THEN
					IF bUseConstantGripTrigger THEN
						rCurrentGripThreshold := aGripScheduleLIVE[1]; 
					ELSE
						rCurrentGripThreshold := aGripScheduleLIVE[nCurrentTestIndex]; 
					END_IF
					
					// Once we've set the value, we can compare to see if we've reached it 
					// Also gate so that the wheel is homed back to the center. 
					IF rGripForce > rCurrentGripThreshold AND ABS(fbEncoder1.rDegrees) < 5 THEN
						bTestIsLive := TRUE; 
					END_IF
					
				END_IF
				
				IF bTestIsLive THEN
					eNextSequenceState := CalibStateType.TEST_ACTIVE; 
					bWheelIsIdle := FALSE; 
					fbTonHoming(IN := bWheelIsIdle); 
					eSetupSubState := HOMING; 
				END_IF
			
			
		END_CASE
		
		
		
		
	// Then we handle logic for actually completing the test. 
	CalibStateType.TEST_ACTIVE: 
	
		// Timer is set based on bTestIsLive variable. Timers are updated at the beginning of every cycle. 	
		IF NOT fbTonPulse.Q THEN // If the pulse hasn't expired, send the pulse 
		
			// We want to split between motor test mode and human test mode. In motor test mode, we artificially add a virtual spring.
			IF NOT bTestTypeHumanLIVE THEN
				
				rAppliedTorque := rConstantTorqueSettingLIVE; 
				rVirtualSpringTorque := -1 * 0.35 * rEncoderRadians;
				// rCommandTorque := rConstantTorqueSettingLIVE - 1 * (0.4 / rAngleNormalizationFactor) * fbEncoder1.rDegrees; 
			ELSE
			
				IF NOT bUseConstantPulseTorque THEN
					rAppliedTorque := 0.4 + 0.02 * rCurrentGripThreshold; 	
				ELSE
					rAppliedTorque := rConstantTorqueSettingLIVE; 
				END_IF
				
				rVirtualSpringTorque := 0;  
			END_IF
			
			rCommandTorque := rAppliedTorque + rVirtualSpringTorque; 
			rCommandVoltage := MotorTorqueToCommandV(rCommandTorque := rCommandTorque); 
			
		ELSE
			IF NOT bTestTypeHumanLIVE THEN 
				rAppliedTorque := 0; 
				rVirtualSpringTorque := -1 * 0.35 * rEncoderRadians;
			ELSE
				rAppliedTorque := 0; 
				rVirtualSpringTorque := 0; 
			END_IF

			rCommandTorque := rAppliedTorque + rVirtualSpringTorque; 
			rCommandVoltage := MotorTorqueToCommandV(rCommandTorque := rCommandTorque); 
		END_IF
		
		fbMotorReference(rCommandVoltage := rCommandVoltage); 
	
		IF fbTonTest.Q THEN
			IF nCurrentTestIndex < UINT_TO_INT(nTrialNumberLIVE) THEN // We have more tests to run 
				bTestIsLive := FALSE;
				nCurrentTestIndex := nCurrentTestIndex + 1; 
				eNextSequenceState := CalibStateType.TEST_SETUP;
			ELSE	
				eNextSequenceState := CalibStateType.TEST_FINISHED; 
				bTestIsLive := FALSE; 
			END_IF
				
		END_IF
		
	
	CalibStateType.TEST_FINISHED: 
		// Start writing to the CSV Then let the log finish. 
		fbLogger.writeLog(); 
		eNextSequenceState := CalibStateType.PROCESSING_LOG; 
		
	CalibStateType.PROCESSING_LOG: 
	
		// We need to check if the processing is still busy
		IF fbLogger.bError THEN
			ADSLOGSTR(
				msgCtrlMask := ADSLOG_MSGTYPE_ERROR OR ADSLOG_MSGTYPE_MSGBOX, 
				msgFmtStr := 'ERROR: Logger has failed during the save process %s', 
				strArg := ''); 
		ELSIF NOT fbLogger.bBusy THEN
			// Now we can reset variabels and go back to the original state. 
			nCurrentTestIndex := 0; 
			nCurrentLaunchIndex := nCurrentLaunchIndex + 1;
			eNextSequenceState := CalibStateType.PRE_LAUNCH; 
		
		END_IF

END_CASE

// Update everything that just happened 
nLastTimeStep := stCalibStepState.nTimestepLow;
fbSystemTime(timeLoDW => stCalibStepState.nTimestepLow, timeHiDW => stCalibStepState.nTimeStepHigh); 
stCalibStepState.rEncoderDegrees := rEncoderDegrees; 
stCalibStepState.rEncoderRadians := rEncoderRadians; 
stCalibStepState.rCommandVoltage := rCommandVoltage; 
stCalibStepState.rCommandTorque := rCommandTorque; 
stCalibStepState.rAppliedTorque := rAppliedTorque; 
stCalibStepState.rVirtualSpringTorque := rVirtualSpringTorque; 
stCalibStepState.rGripForce := rGripForce; 
stCalibStepState.rCurrentGripThreshold := rCurrentGripThreshold; 
stCalibStepState.sSequenceStateString := TO_STRING(eSequenceState); 
stCalibStepState.nCurrentTestIndex := nCurrentTestIndex; 
stCalibStepState.nTestIsLive := BOOL_TO_INT(bTestIsLive); 

// If we're in the setup or active phase, we add it to the log. 
IF eSequenceState = CalibStateType.TEST_ACTIVE THEN
	fbLogger.addStep(stNewStep := stCalibStepState); 
END_IF

// Update state for next iteration
eSequenceState := eNextSequenceState; 

GVL.ENCODER_1_COUNTER_VALUE := nEncoderCounts; 
GVL.ENCODER_1_DEGREES := rEncoderDegrees; 
GVL.MOTOR_1_APPLIED_VOLTAGE := rCommandVoltage;
GVL.LOAD_CELL_NEWTONS := rGripForce; 
GVL.CALIB_SYSTEM_TIME := stCalibStepState.nTimestepLow - nLastTimeStep;

METHOD Reset : BOOL
VAR_INPUT
END_VAR
fbEncoder1.Reset();
END_METHOD

END_FUNCTION_BLOCK

// ---- POUs/MetadataBlock.TcPOU
FUNCTION_BLOCK MetadataBlock
VAR_INPUT
END_VAR
VAR_OUTPUT
	bBusy : BOOL := FALSE; 
	bError : BOOL := FALSE; 
	sUserID : STRING(400) := ''; 
END_VAR
VAR
	bGenerateRandomID : BOOL := TRUE; 
	drand : DRAND; 
	rRandomIDFloat : LREAL; 
	nRandomID : DINT; 
	sFilename : STRING(400) := ''; 
	sDescriptionBox : STRING(1000); 
	sNotesBox : STRING(1000); 
	
	// File writing variables
	sDefaultDirectory : T_MaxString := 'C:\Users\njanne\Documents\DDTestLogs\metadata\';
	bWriteToDisk : BOOL := FALSE; 
	bIDWritten : BOOL := FALSE; 
	bDescWritten : BOOL := FALSE; 
	bNotesWritten : BOOL := FALSE; 
	nFileHandle : UINT; 
	eFileWriteState : (IDLE, OPEN, WRITE, CLOSE, ERROR); 
	nFileWriteSubstep : INT := 0; 
	sTempString : STRING(1000); 
	sNewline : STRING := '$n'; 
	
	// Helper function blocks
	fbFormatString : FB_FormatString; 
	fbFormatString2 : FB_FormatString2; 
	fbFileOpen : FB_FileOpen; 
	fbFilePuts : FB_FilePuts; 
	fbFileClose : FB_FileClose; 
	
END_VAR

IF bGenerateRandomID THEN 
	drand(Num => rRandomIDFloat); 
	rRandomIdFloat := rRandomIDFloat * 1000000; 
	nRandomID := LREAL_TO_DINT(rRandomIDFloat); 
	fbFormatString(sFormat := '%06d', arg1 := F_DINT(nRandomID)); 
	sUserID := fbFormatString.sOut; 
	bGenerateRandomID := FALSE; 
END_IF

IF bWriteToDisk THEN 
	
	// If it's time to write to disk, we need to empty the buffer. 
	CASE eFileWriteState OF 
		
		IDLE: 
			// Get everything read. 
			fbFormatString(sFormat := '%s.txt', arg1 := F_STRING(sUserId)); 
			sFilename := fbFormatString.sOut; 
			nFileHandle := 0; 
			bBusy := TRUE; 
			eFileWriteState := OPEN; 
			nFileWriteSubstep := 0; 
	
		OPEN: 
			CASE nFileWriteSubstep OF 
				0: 
					// Opens a file for writing at the end of the file 
					fbFileOpen(sPathName := CONCAT(sDefaultDirectory, sFilename), bExecute := FALSE); 
					fbFileOpen(
						bExecute		:= TRUE, 
						sNetID			:= '', 
						sPathName		:= CONCAT(sDefaultDirectory, sFilename),
						nMode 			:= FOPEN_MODEAPPEND OR FOPEN_MODETEXT); 
						
					nFileWriteSubstep := nFileWriteSubstep + 1; // Advance to wait for open. 
					
				1: 
					fbFileOpen(bExecute := FALSE); 
					IF NOT fbFileOpen.bBusy THEN 
						IF fbFileOpen.bError THEN 
							eFileWriteState := ERROR; 
							nFileWriteSubstep := 0; 
						ELSE 
							nFileHandle := fbFileOpen.hFile; 
							eFileWriteState := WRITE; 
							nFileWriteSubstep := 0;
						END_IF
					END_IF
			END_CASE
			
		WRITE: 
			CASE nFileWriteSubstep OF 
				0 : 
					fbFilePuts(bExecute := FALSE); 
					
					// Check if we need to write the ID 
					IF NOT bIDWritten THEN 
						CONCAT2(ADR(sFilename), ADR(sNewline), pDstString := ADR(sTempString), nDstSize := SIZEOF(sTempString)); 
						bIDWritten := TRUE; 
					ELSIF NOT bDescWritten THEN 
						CONCAT2(ADR(sDescriptionBox), ADR(sNewline), pDstString := ADR(sTempString), nDstSize := SIZEOF(sTempString));
						bDescWritten := TRUE; 
					ELSIF NOT bNotesWritten THEN
						CONCAT2(ADR(sNotesBox), ADR(sNewline), pDstString := ADR(sTempString), nDstSize := SIZEOF(sTempString));
						bNotesWritten := TRUE; 
					END_IF
			
					fbFilePuts(
						bExecute		:= TRUE, 
						sNetID			:= '', 
						hFile			:= nFileHandle, 
						sLine			:= sTempString); 
					
					nFileWriteSubstep := nFileWriteSubstep + 1; 
					
				1 : 
					fbFilePuts(bExecute := FALSE); 
					IF NOT fbFilePuts.bBusy THEN 
						IF fbFilePuts.bError THEN 
							eFileWriteState := ERROR; 
							nFileWriteSubstep := 0; 
						ELSE 
							// Check if we have more things to write 
							IF bNotesWritten THEN 
								eFileWriteState := CLOSE;
							ELSE 
								eFileWriteState := WRITE;
							END_IF
						END_IF
						nFileWriteSubstep := 0; 
					END_IF

			END_CASE
			
		CLOSE: 
			CASE nFileWriteSubstep OF 
				0: 
					fbFileClose(bExecute := FALSE); 
					fbFileClose(
						bExecute		:= TRUE,
						sNetId			:= '', 
						hFile			:= nFileHandle); 
					nFileWriteSubstep := nFileWriteSubstep + 1; 
				1: 
					fbFileClose(bExecute := FALSE); 
					IF NOT fbFileClose.bBusy THEN 
						IF fbFileClose.bError THEN 
							eFileWriteState := ERROR; 
							nFileWriteSubstep := 0; 
						ELSE
							eFileWriteState := IDLE; 
							nFileHandle := 0; 
							
							// Also reset everything so taht a new file can be written 
							nFileWriteSubstep := 0; 
							bIDWritten := FALSE; 
							bDescWritten := FALSE; 
							bNotesWritten := FALSE; 
							bBusy := FALSE; 
							bWriteToDisk := FALSE; 
							
						END_IF
					END_IF
			END_CASE
			
		ERROR: 
			// Error, clear the handle and go back to idle. 
			nFileHandle := 0;
			eFileWriteState := IDLE; 
			bError := TRUE; 
	
	END_CASE

END_IF

END_FUNCTION_BLOCK

// ---- POUs/MAIN.TcPOU
PROGRAM MAIN
VAR
	
	// Establish state machine for hardware
	MASTER_STATE : MasterStateType := MasterStateType.WAITING;
	PREVIOUS_MASTER_STATE : MasterStateType := MasterStateType.WAITING; 
	MASTER_STATE_STR : STRING := TO_STRING(MASTER_STATE);

	// Establish state machine for GUI
	WINDOW_STATE : ActiveWindowStateType := ActiveWindowStateType.EXPERIMENT_WINDOW; 
	
	// Load submodules 
	fbMainExperimentBlock : MainExperimentBlock; 
	fbCalibrationBlock : CalibrationBlock;
	fbWaitingMonitorBlock : WaitingMonitorBlock;
	
	// Motor commands (and other outputs), need to be commanded 
	// by a top level function if multiple objects are going to control it. 
	fbMotor1 : FB_AnalogMotorDriver; 
	fbSystemTime : GETSYSTEMTIME; 
	Metablock : MetadataBlock; 
	
END_VAR

// Update system time
fbSystemTime(timeLoDW => GVL.MAIN_SYSTEM_TIME); 

// Update any metadata 
Metablock(); 

// Update master state string to send to GUI 
MASTER_STATE_STR := TO_STRING(MASTER_STATE);

// Based on the master state, load different behavior profile. 
// Check to make sure that we reset a block's behavior after leaving it.
IF PREVIOUS_MASTER_STATE = MasterStateType.ACTIVE AND MASTER_STATE <> MasterStateType.ACTIVE THEN
	fbMainExperimentBlock.Reset(); 
	fbMotor1.Reset(); 
END_IF
IF PREVIOUS_MASTER_STATE = MasterStateType.CALIBRATION AND MASTER_STATE <> MasterStateType.CALIBRATION THEN
	fbCalibrationBlock.Reset();
	fbMotor1.Reset(); 
END_IF
IF PREVIOUS_MASTER_STATE = MasterStateType.WAITING AND MASTER_STATE <> MasterStateType.WAITING THEN
	fbWaitingMonitorBlock.Reset();
	fbMotor1.Reset();
END_IF

CASE MASTER_STATE OF
	MasterStateType.ACTIVE : 
		fbMainExperimentBlock(fbMotorReference := fbMotor1, fbMetadata := Metablock);
 
	MasterStateType.CALIBRATION : 
		fbCalibrationBlock(fbMotorReference := fbMotor1, fbMetadata := Metablock);
	
	MasterStateType.WAITING: 
		fbWaitingMonitorBlock(fbMotorReference := fbMotor1, fbMetadata := Metablock);
END_CASE

// Update previous master state, recall master state 
// itself is controlled by GUI
PREVIOUS_MASTER_STATE := MASTER_STATE;

END_PROGRAM

// ---- POUs/MainExperimentBlock.TcPOU
FUNCTION_BLOCK MainExperimentBlock
VAR_INPUT

	fbMotorReference : REFERENCE TO FB_AnalogMotorDriver; 
	fbMetadata : REFERENCE TO MetadataBlock; 

END_VAR
VAR_OUTPUT

	// Variables for logging
	nEncoderCounts : LINT; 
	rEncoderDegrees : REAL;
	rEncoderLastDegrees : REAL; 
	rEncoderRadians : REAL; 
	rEncoderLastRadians : REAL; 
	rEncoderRadiansBuffer : ARRAY[1..FILTER_WINDOW] OF REAL; 
	rEncoderRadiansSum : REAL; 
	rEncoderRadiansFiltered : REAL; 
	nFilterBufferCount : INT := 0; 

	// Variables for motor control 
	rCommandVoltage : REAL; 
	rCommandTorque : REAL; 
	rError : REAL; 
	rLastError : REAL; 
	rProportional : REAL; 
	rIntegral : REAL := 0; 
	rDerivative : REAL; 
	bPIDStale : BOOL := TRUE;
	rControlOutput : REAL; 
	Kp : REAL := 0.3; 
	Ki : REAL := 0.03; 
	Kd : REAL := 0.05; 
	d_time : REAL := 0.0001; // Time step (100 us). 
	
	// Variables for load cell 
	rGripForce : REAL; 

END_VAR
VAR CONSTANT
	nMaxTestNumber : INT := 10; 

	// Load constants (for virtual wall) 
	aLOAD_CONSTANTS : ARRAY[1..5] OF REAL := [0.1, 0.2, 0.3, 0.4, 0.5]; 
	
	// Constants for digital filtering 
	FILTER_WINDOW : INT := 11; 
	
END_VAR
VAR
	
	// Variables to keep track of the actual encoder/motor setup 
	fbEncoder1 : FB_QuadratureEncoder;
	fbLoadCell : FB_AnalogLoadCellInput; 
	rNormalizedWheelPosition : REAL; 
	
	// Settings to manage experiment behavior.  
	eSequenceState : MainStateType := MainStateType.PRE_LAUNCH; 
	eNextSequenceState : MainStateType := MainStateType.PRE_LAUNCH;
	stMainStepState : ST_MainTrialStep;  
	eSetupSubState : (HOMING, WAITING); 
	nCurrentTestIndex : INT := 0; 
	nCurrentLaunchIndex : INT := 0; 
	bLaunchTestSequence : BOOL := FALSE; 
	bTestIsLive : BOOL := FALSE; 
	nTestIsLive : INT; 
	bDemoMode : BOOL := FALSE; 
	nDemoLoadSetting : INT := 1; 
	aTestSettings : ARRAY[1..nMaxTestNumber] OF ST_LoadExperimentSetting; 
	bInitTestSettings : BOOL := FALSE; 
	bInitHLCatch : BOOL := FALSE; // Implement Heavy-Light Catch
	bInitLHCatch : BOOL := FALSE; // Implement Light-Heavy Catch
	bInitExtrap : BOOL := FALSE; // Implement Random Extrapolation
	binitInterp : BOOL := FALSE; // Implement Random Interpolation
		
	// Intermediate variables for virtual spring
	rAngleThreshold : REAL := LREAL_TO_REAL(DEG_TO_RAD(80)); 
	
	rAngleTarget : REAL := LREAL_TO_REAL(DEG_TO_RAD(60)); 
	rAngleTargetRange : REAL := LREAL_TO_REAL(DEG_TO_RAD(8)); 
	bTargetIsInRange : BOOL := FALSE; 
	
	
	rStartGripThreshold : REAL := 1.5; // Threshold to start the test (amount of force required by hand). 

	// Helpers 
	i : INT; 
	j : INT; 
	TempString : T_MaxString; 
	bWheelIsIdle : BOOL; 
	fbTonHoming : TON := (PT := T#500MS); // Time to give state machine to home
	fbTonTargetReached : TON := (PT := T#1000MS); // Time where subject should hold wheel in target position.
	
	drand : DRAND; 
	rRand : LREAL; // Random variable. 
	fbSystemTime : GETSYSTEMTIME; 
	fbFormatString : FB_FormatString; 
	fbLogger : MainExperimentBlockLogger; 
	
END_VAR

// Initialize settings array if need be 
IF NOT bInitTestSettings THEN
	FOR i := 1 TO nMaxTestNumber DO
		aTestSettings[i].Test_Finished := FALSE; 
		aTestSettings[i].Weight := 1;
	END_FOR
	bInitTestSettings := TRUE; 
END_IF
IF bInitHLCatch THEN 
	FOR i := 1 TO nMaxTestNumber DO 
		aTestSettings[i].Test_Finished := FALSE; 
		aTestSettings[i].Weight := 4;
	END_FOR	
	
	// Generate random place to start light case
	drand(Num => rRand); 
	
	// Start index 
	j := LREAL_TO_INT(rRand * 6 + 3);

	FOR i := j TO nMaxTestNumber DO
		aTestSettings[i].Weight := 2; 
	END_FOR 
	bInitHLCatch := FALSE; 
END_IF
IF bInitLHCatch THEN
	FOR i := 1 TO nMaxTestNumber DO 
		aTestSettings[i].Test_Finished := FALSE; 
		aTestSettings[i].Weight := 2; 
	END_FOR
	
	// Generate random video to start light case
	drand(Num => rRand); 
	
	// Start index 
	j := LREAL_TO_INT(rRand * 6 + 3); 
	
	FOR i := j TO nMaxTestNumber DO 
		aTestSettings[i].Weight := 4; 
	END_FOR
	bInitLHCatch := FALSE; 
END_IF

// Read sensors on current iteration

// Encoders 
fbEncoder1(); 
nEncoderCounts := fbEncoder1.nNetCounts; 
rEncoderDegrees := fbEncoder1.rDegrees; 
rEncoderLastDegrees := fbEncoder1.rLastDegrees; 
rEncoderRadians := fbEncoder1.rRadians; 
rEncoderLastRadians := fbEncoder1.rLastRadians;

// Update digital filter. 
IF nFilterBufferCount < FILTER_WINDOW THEN 
	nFilterBufferCount := nFilterBufferCount + 1; 
END_IF

// Shift the buffer and add the new reading 
FOR i := FILTER_WINDOW TO 2 BY -1 DO
	rEncoderRadiansBuffer[i] := rEncoderRadiansBuffer[i-1]; 
END_FOR
rEncoderRadiansBuffer[1] := rEncoderRadians;

// Computer the moving average only if the buffer is full
j := MIN(nFilterBufferCount, FILTER_WINDOW); 
rEncoderRadiansSum := 0.0; 
FOR i:= 1 TO j DO
	rEncoderRadiansSum := rEncoderRadiansSum + rEncoderRadiansBuffer[i];
END_FOR
rEncoderRadiansFiltered := rEncoderRadiansSum / j; 


// Load cell 
fbLoadCell(); 
rGripForce := fbLoadCell.rCalibratedOutput; 


// Now we check to see if we're in demo mode, or we're in a live testing mode. 
IF bDemoMode THEN

	// Apply the standard virtual wall condition. 
	rNormalizedWheelPosition := rEncoderRadians / 0.1; 
	
	IF rNormalizedWheelPosition > 1 THEN
		rCommandTorque := -1 * aLOAD_CONSTANTS[nDemoLoadSetting]; 
		rCommandVoltage := MotorTorqueToCommandV(rCommandTorque := rCommandTorque);
	ELSIF rNormalizedWheelPosition > 0 THEN
		rCommandTorque := -1 * rNormalizedWheelPosition * aLOAD_CONSTANTS[nDemoLoadSetting]; 
		rCommandVoltage := MotorTorqueToCommandV(rCommandTorque := rCommandTorque);	
	ELSE
		rCommandTorque := 0; 
		rCommandVoltage := 0;
	END_IF
	
	// Then send command to the motor. 
	fbMotorReference(rCommandVoltage := rCommandVoltage); 
	

ELSE

	// Generate the file name and update the logger. 
	fbFormatString(
		sFormat := '%s_test_%d.csv', 
		arg1 := F_STRING(fbMetadata.sUserID), 
		arg2 := F_INT(nCurrentLaunchIndex));
		
	fbLogger(sFileName := fbFormatString.sOut); 
	

	// In the live testing mode, we're running through the state machine. 
	CASE eSequenceState OF
		
		MainStateType.PRE_LAUNCH: 
		
			// First we start by updating options
			IF bLaunchTestSequence THEN 
				eNextSequenceState := MainStateType.TEST_SETUP; 
				eSetupSubState := HOMING; 
				
				// Also set the first test index 
				nCurrentTestIndex := 1; 
				
				// And put this signal back down 
				bLaunchTestSequence := FALSE; 
				
			ELSE
				eNextSequenceState := MainStateType.PRE_LAUNCH; 
			END_IF
			
			// We also need to make sure any motor commands are no longer hanging over 
			bTestIsLive := FALSE; 
			rCommandTorque := 0; 
			rCommandVoltage := 0; 
			fbMotorReference(rCommandVoltage := rCommandVoltage); 
	
		// We are getting the test ready. 
		MainStateType.TEST_SETUP: 
		
			CASE eSetupSubState OF
				
				HOMING: 
				
					// In this state, we need to recenter the motor back to the 0 point, and 
					// we also need to wait for the triggering signal. 
					rError := 0 - rEncoderRadiansFiltered; 
					rProportional := Kp * rError; 
					rIntegral := rIntegral + (rError * d_time); 
					rDerivative := (rError - rLastError) / d_time; 
					rLastError := rError; 
					//rCommandTorque := -1 * ((3/2) * rEncoderRadians - (2/3) * rEncoderLastRadians);
					IF bPIDStale THEN
						rCommandTorque := rProportional;
						rIntegral := 0; 
						bPIDStale := FALSE; 
					ELSE 
						rCommandTorque := rProportional + (Ki * rIntegral) + (Kd * rDerivative);
					END_IF
					rCommandVoltage := MotorTorqueToCommandV(rCommandTorque := rCommandTorque); 
					fbMotorReference(rCommandVoltage := rCommandVoltage); 
					
					// Check to see if the wheel has been idle for long enough. 
					bWheelIsIdle := rGripForce < rStartGripThreshold AND ABS(rEncoderDegrees) < 5;  
					fbTonHoming(IN := bWheelIsIdle); 
					
					IF fbTonHoming.Q THEN
						eSetupSubState := WAITING; 
					END_IF
					
				WAITING:
					IF rGripForce > rStartGripThreshold THEN
						bTestIsLive := TRUE; 
						eNextSequenceState := MainStateType.TEST_ACTIVE; 
						bWheelIsIdle := FALSE; 
						fbTonHoming(IN := bWheelIsIdle); 
						eSetupSubState := HOMING; 
					END_IF 
					
			END_CASE
		
		// Handle logic for actually completing the test. 
		MainStateType.TEST_ACTIVE: 
			
			// Apply the standard virtual wall condition. 
			rNormalizedWheelPosition := rEncoderRadians / 0.1; 
			
			IF rNormalizedWheelPosition > 1 THEN
				rCommandTorque := -1 * aLOAD_CONSTANTS[aTestSettings[nCurrentTestIndex].Weight]; 
				rCommandVoltage := MotorTorqueToCommandV(rCommandTorque := rCommandTorque);
			ELSIF rNormalizedWheelPosition > 0 THEN
				rCommandTorque := -1 * rNormalizedWheelPosition * aLOAD_CONSTANTS[aTestSettings[nCurrentTestIndex].Weight]; 
				rCommandVoltage := MotorTorqueToCommandV(rCommandTorque := rCommandTorque);	
			ELSE
				rCommandTorque := 0; 
				rCommandVoltage := 0;
			END_IF
			
			// Then send command to the motor. 
			fbMotorReference(rCommandVoltage := rCommandVoltage);
			
			// Check to see if we need to get out of this state (test is finished)
			bTargetIsInRange := ABS(rEncoderradians - rAngleTarget) <= rAngleTargetRange; 
			fbTonTargetReached(IN := bTargetIsInRange); 
			
			IF fbTonTargetReached.Q THEN // Trial is complete 
				aTestSettings[nCurrentTestIndex].Test_Finished := TRUE; 
				bTestIsLive := FALSE; 
				eNextSequenceState := MainStateType.WAITING_FOR_RELEASE; 
			END_IF
 
//			IF rEncoderRadians > rAngleThreshold THEN
//				aTestSettings[nCurrentTestIndex].Test_Finished := TRUE; 
//				bTestIsLive := FALSE; 
		
//				eNextSequenceState := MainStateType.WAITING_FOR_RELEASE; 
				
//			END_IF
			

		MainStateType.WAITING_FOR_RELEASE: // Wait for the user to drop the wheel
		
			bWheelIsIdle := rGripForce < rStartGripThreshold; 
			fbTonHoming(IN := bWheelIsIdle);
		
			IF fbTonHoming.Q THEN
				// There's more tests to run! 
				IF nCurrentTestIndex < nMaxTestNumber THEN
					nCurrentTestIndex := nCurrentTestIndex + 1; 
					eNextSequenceState := MainStateType.TEST_SETUP; 
					bPIDStale := TRUE; 
				ELSE
					eNextSequenceState := MainStateType.TEST_FINISHED; 
				END_IF
				
				// Reset the timer 
				bWheelIsIdle := FALSE; 
				fbTonHoming(IN := bWheelIsIdle); 
				
			ELSE
				eNextSequenceState := MainStateType.WAITING_FOR_RELEASE; 
			END_IF
			
			rCommandTorque := 0; 
			rCommandVoltage := 0; 
			fbMotorReference(rCommandVoltage := rCommandVoltage); 
			
		MainStateType.TEST_FINISHED: 
			// trigger log writing. 
			fbLogger.writeLog(); 
			eNextSequenceState := MainStateType.PROCESSING_LOG; 
			
			
		MainStateType.PROCESSING_LOG: 
		
			// We need to check if the processing is still busy 
			IF fbLogger.bError THEN
				ADSLOGSTR(
					msgCtrlMask := ADSLOG_MSGTYPE_ERROR OR ADSLOG_MSGTYPE_MSGBOX,
					msgFmtStr := 'ERROR: Logger has failed during the save process %s', 
					strArg := ''); 
			ELSIF NOT fbLogger.bBusy THEN
				// Check for errors, then go back to pre-launch 
				nCurrentTestIndex := 0; 
				nCurrentLaunchIndex := nCurrentLaunchIndex + 1; 
				eNextSequenceState := MainStateType.PRE_LAUNCH; 
			END_IF
			
	END_CASE

	// Update logs 
	// Check whether or not to post to the log. 
	IF nCurrentTestIndex > 0 THEN
		fbSystemTime(timeLoDW => stMainStepState.nTimestepLow, timeHiDW => stMainStepState.nTimestepHigh);
		stMainStepState.rEncoderDegrees := rEncoderDegrees; 
		stMainStepState.rEncoderRadians := rEncoderRadians;
		stMainStepState.rCommandVoltage := rCommandVoltage; 
		stMainStepState.rCommandTorque := rCommandTorque; 
		stMainStepState.rWallTorque := aLOAD_CONSTANTS[aTestSettings[nCurrentTestIndex].Weight];
		stMainStepState.rGripForce := rGripForce; 
		stMainStepState.sSequenceStateString := TO_STRING(eSequenceState); 
		stMainStepState.nCurrentTestIndex := nCurrentTestIndex; 
		stMainStepState.nTestIsLive := BOOL_TO_INT(bTestIsLive); 
	END_IF
	
	IF eSequenceState = MainStateType.TEST_ACTIVE THEN
		// Push the step to the log. 
		fbLogger.addStep(stNewStep := stMainStepState); 
	END_IF
	
	// Update state for next iteration. 
	eSequenceState := eNextSequenceState; 
	

END_IF

// Update globals for logging 
GVL.ENCODER_1_COUNTER_VALUE := nEncoderCounts; 
GVL.ENCODER_1_DEGREES := rEncoderDegrees;
GVL.MOTOR_1_APPLIED_VOLTAGE := rCommandVoltage; 
GVL.LOAD_CELL_NEWTONS := rGripForce;

METHOD Reset : BOOL
VAR_INPUT
END_VAR
fbEncoder1.Reset();
END_METHOD

END_FUNCTION_BLOCK

// ---- POUs/MainExperimentBlockLogger.TcPOU
FUNCTION_BLOCK MainExperimentBlockLogger
VAR_INPUT
	sFileName : STRING; 
END_VAR
VAR_OUTPUT
	bBusy : BOOL := FALSE; 
	bError : BOOL := FALSE; 
END_VAR
VAR CONSTANT
	nMaxBufferSize : UDINT := 2000000;
END_VAR
VAR
	cDefaultHeader : T_MaxString := 'TimeLow,TimeHigh,EncoderDegrees,EncoderRadians,CommandVoltage,CommandTorque,WallTorque,GripForce,SequenceState,CurrentTestIndex,TestIsLive $n'; 
	sDefaultDirectory : T_MaxString := 'C:\Users\njanne\Documents\DDTestLogs\main\';
	bWriteToDisk : BOOL := FALSE; 
	eFileWriteState : (IDLE, OPEN, WRITE, CLOSE, ERROR); 
	nFileWriteSubstep : INT := 0; 
	fbFileOpen : FB_FileOpen; 
	fbFilePuts : FB_FilePuts; 
	fbFileClose : FB_FileClose; 
	fbFormatString : FB_FormatString2; 
	nFileHandle : UINT; 
	bHeaderWriteComplete : BOOL := FALSE; 
	nWriteIndex : UDINT := 0; 
	sWritePercentFormat : T_MaxString := '%.2f %%'; 
	rWritePercent : REAL; 
	sWritePercentString : T_MaxString; 
	
	// For formatting data into a string. 
	sDataFormatStr1 : STRING := '%d,%d,%f,%f,%f,%f,%f,%f,%s,%d,'; 
	sDataFormatStr2 : STRING := '%d $n';
	sTempString : STRING(600); 
	sOutputString : STRING(600); 
	
	// For data storage 
	aTrialDataBuffer : ARRAY[0..nMaxBufferSize] OF ST_MainTrialStep; 
	nStepsSoFar : UDINT := 0;  // Current number of steps in the database. 
	
END_VAR

IF bWriteToDisk THEN 
	

	// If it's time to write to disk, we need to empty the buffer. 
	CASE eFileWriteState OF 
		
		IDLE: 
			// Get everything ready. 
			nFileHandle := 0; 
			bBusy := TRUE; 
			eFileWriteState := OPEN; 
			nFileWriteSubstep := 0; 
			
		OPEN: 
			CASE nFileWriteSubstep OF 
				0: 
					// Opens a file for writing at the end of the file (append). 
					// if the file does not exist, a new file is created. 
					fbFileOpen(sPathName := CONCAT(sDefaultDirectory, sFilename), bExecute := FALSE); 
					fbFileOpen(
						bExecute		:= TRUE, 
						sNetID			:= '', 
						sPathName		:= CONCAT(sDefaultDirectory, sFilename),
						nMode 			:= FOPEN_MODEAPPEND OR FOPEN_MODETEXT); 
						
					nFileWriteSubstep := nFileWriteSubstep + 1; // Advance to wait for open. 
				
				1: 
					fbFileOpen(bExecute := FALSE); 
					IF NOT fbFileOpen.bBusy THEN
						IF fbFileOpen.bError THEN 
							eFileWriteState := ERROR; 
							nFileWriteSubstep := 0; 
						ELSE
							nFileHandle := fbFileOpen.hFile; 
							eFileWriteState := WRITE; 
							nFileWriteSubstep := 0; 
						END_IF
					END_IF
				END_CASE
				
			WRITE: 
				CASE nFileWriteSubstep OF 
					0 : 
						fbFilePuts(bExecute := FALSE); 
						
						// Check if we still need to write the header. 
						IF NOT bHeaderWriteComplete THEN 
							fbFilePuts(
								bExecute		:= TRUE, 
								sNetId			:= '', 
								hFile			:= nFileHandle, 
								sLine			:= cDefaultHeader); 
							bHeaderWriteComplete := TRUE; 
						ELSE
							// If the header is already written, then we're going for data. 
							// We need to first format the string. 
							fbFormatString(
								pFormatString := ADR(sDataFormatStr1), 
								arg1 := F_UDINT(aTrialDataBuffer[nWriteIndex].nTimestepLow), 
								arg2 := F_UDINT(aTrialDataBuffer[nWriteIndex].nTimestepHigh), 
								arg3 := F_REAL(aTrialDataBuffer[nWriteIndex].rEncoderDegrees), 
								arg4 := F_REAL(aTrialDataBuffer[nWriteIndex].rEncoderRadians), 
								arg5 := F_REAL(aTrialDataBuffer[nWriteIndex].rCommandVoltage), 
								arg6 := F_REAL(aTrialDataBuffer[nWriteIndex].rCommandTorque), 
								arg7 := F_REAL(aTrialDataBuffer[nWriteIndex].rWallTorque), 
								arg8 := F_REAL(aTrialDataBuffer[nWriteIndex].rGripForce), 
								arg9 := F_STRING(aTrialDataBuffer[nWriteIndex].sSequenceStateString), 
								arg10 := F_INT(aTrialDataBuffer[nWriteIndex].nCurrentTestIndex), 
								pDstString := ADR(sOutputString), 
								nDstSize := SIZEOF(sOutputString)); 
							
							fbFormatString(
								pFormatString := ADR(sDataFormatStr2), 
								arg1 := F_INT(aTrialDataBuffer[nWriteIndex].nTestIsLive), 
								pDstString := ADR(sTempString), 
								nDstSize := SIZEOF(sTempString)); 
								
							CONCAT2(
								pSrcString1 := ADR(sOutputString), 
								pSrcString2 := ADR(sTempString), 
								pDstString := ADR(sOutputString), 
								nDstSize := SIZEOF(sOutputString));
								
							fbFilePuts(
								bExecute		:= TRUE, 
								sNetId			:= '', 
								hFile			:= nFileHandle,
								sLine			:= sOutputString); 

							// Update write progress
							nWriteIndex := nWriteIndex + 1; 
							rWritePercent := UDINT_TO_REAL(nWriteIndex) / UDINT_TO_REAL(nStepsSoFar) * 100; 
							fbFormatString(
								pFormatString := ADR(sWritePercentFormat), 
								arg1 := F_REAL(rWritePercent), 
								pDstString := ADR(sWritePercentString), 
								nDstSize := SIZEOF(sWritePercentString)); 
							
						END_IF
						
						nFileWriteSubstep := nFileWriteSubstep + 1; // Advance to waiting state. 
						
					1 : 
						fbFilePuts(bExecute := FALSE); 
						IF NOT fbFilePuts.bBusy THEN 
							IF fbFilePuts.bError THEN 
								eFileWriteState := ERROR; 
								nFileWriteSubstep := 0; 
							ELSE 
								// Check if we have more things to write to the file. 
								IF nWriteIndex = nStepsSoFar THEN 
									eFileWriteState := CLOSE; 
								ELSE 
									eFileWriteState := WRITE; 
								END_IF
							END_IF
							nFileWriteSubstep := 0; 
						END_IF
						
				END_CASE
				
			CLOSE: 
				CASE nFileWriteSubstep OF 
					0:
						fbFileClose(bExecute := FALSE); 
						fbFileClose(
							bExecute		:= TRUE, 
							sNetId			:= '', 
							hFile			:= nFileHandle); 
						nFileWriteSubstep := nFileWriteSubstep + 1; 
						
					1: 
						fbFileClose(bExecute := FALSE); 
						IF NOT fbFileClose.bBusy THEN 
							IF fbFileClose.bError THEN 
								eFileWriteState := ERROR; 
								nFileWriteSubstep := 0; 
							ELSE
								eFileWriteState := IDLE; 
								nFileHandle := 0;
								
								// Also reset everything so that a new file can be written. 
								nStepsSoFar := 0; 
								nWriteIndex := 0; 
								nFileWriteSubstep := 0; 
								bHeaderWriteComplete := FALSE; 
								bBusy := FALSE; 
								bWriteToDisk := FALSE;
							END_IF
						END_IF
					END_CASE
						
			ERROR: 
				// Error, clear the handle and go back to idle. 
				nFileHandle := 0; 
				eFileWriteState := IDLE; 
				bError := TRUE; 
	
	END_CASE

END_IF

METHOD addStep : BOOL
VAR_INPUT
	stNewStep : ST_MainTrialStep; // The incoming step to be added to memory
END_VAR
// We need to simply copy over all the fields into the new position. 
// And then, update the counter. 
MEMCPY(
	destAddr := ADR(aTrialDataBuffer[nStepsSoFar]), 
	srcAddr := ADR(stNewStep), 
	n := SIZEOF(ST_MainTrialStep)); 
	
nStepsSoFar := nStepsSoFar + 1;
END_METHOD

METHOD writeLog : BOOL
VAR_INPUT
END_VAR
bWriteToDisk := TRUE;
END_METHOD

END_FUNCTION_BLOCK

// ---- POUs/WaitingMonitorBlock.TcPOU
FUNCTION_BLOCK WaitingMonitorBlock
VAR_INPUT

	fbMotorReference : REFERENCE TO FB_AnalogMotorDriver; 
	fbMetadata : REFERENCE TO MetadataBlock; 

END_VAR
VAR_OUTPUT

	// Variables for logging
	nEncoderCounts : LINT; 
	rEncoderDegrees : REAL;
	rEncoderLastDegrees : REAL; 
	rEncoderRadians : REAL; 
	rEncoderLastRadians : REAL; 
	rEncoderRadiansBuffer : ARRAY[1..FILTER_WINDOW] OF REAL; 
	rEncoderRadiansSum : REAL; 
	rEncoderRadiansFiltered : REAL; 
	nFilterBufferCount : INT := 0; 

	// Variables for motor control 
	rCommandVoltage : REAL; 
	rCommandTorque : REAL; 
	rError : REAL; 
	rLastError : REAL; 
	rProportional : REAL; 
	rIntegral : REAL := 0; 
	rDerivative : REAL; 
	bPIDStale : BOOL := TRUE;
	rControlOutput : REAL; 
	Kp : REAL := 0.3; 
	Ki : REAL := 0.03; 
	Kd : REAL := 0.05; 
	d_time : REAL := 0.0001; // Time step (100 us). 
	
	// Variables for load cell 
	rGripForce : REAL; 

END_VAR
VAR CONSTANT
	nMaxTestNumber : INT := 10; 

	// Load constants (for virtual wall) 
	aLOAD_CONSTANTS : ARRAY[1..5] OF REAL := [0.1, 0.2, 0.3, 0.4, 0.5]; 
	
	// Constants for digital filtering 
	FILTER_WINDOW : INT := 11; 
	
END_VAR
VAR
	
	// Variables to keep track of the actual encoder/motor setup 
	fbEncoder1 : FB_QuadratureEncoder;
	fbLoadCell : FB_AnalogLoadCellInput; 
	rNormalizedWheelPosition : REAL; 
		
	// Intermediate variables for virtual spring
	rAngleThreshold : REAL := LREAL_TO_REAL(DEG_TO_RAD(80)); 
	
	rAngleTarget : REAL := LREAL_TO_REAL(DEG_TO_RAD(60)); 
	rAngleTargetRange : REAL := LREAL_TO_REAL(DEG_TO_RAD(8)); 
	bTargetIsInRange : BOOL := FALSE; 
	
	
	rStartGripThreshold : REAL := 1.5; // Threshold to start the test (amount of force required by hand). 

	// Helpers 
	i : INT; 
	j : INT; 
	TempString : T_MaxString; 
	bWheelIsIdle : BOOL; 
	fbTonHoming : TON := (PT := T#500MS); // Time to give state machine to home
	fbTonTargetReached : TON := (PT := T#1000MS); // Time where subject should hold wheel in target position.
	
END_VAR

// Encoders 
fbEncoder1(); 
nEncoderCounts := fbEncoder1.nNetCounts; 
rEncoderDegrees := fbEncoder1.rDegrees; 
rEncoderLastDegrees := fbEncoder1.rLastDegrees; 
rEncoderRadians := fbEncoder1.rRadians; 
rEncoderLastRadians := fbEncoder1.rLastRadians;

// Update digital filter. 
IF nFilterBufferCount < FILTER_WINDOW THEN 
	nFilterBufferCount := nFilterBufferCount + 1; 
END_IF

// Shift the buffer and add the new reading 
FOR i := FILTER_WINDOW TO 2 BY -1 DO
	rEncoderRadiansBuffer[i] := rEncoderRadiansBuffer[i-1]; 
END_FOR
rEncoderRadiansBuffer[1] := rEncoderRadians;

// Computer the moving average only if the buffer is full
j := MIN(nFilterBufferCount, FILTER_WINDOW); 
rEncoderRadiansSum := 0.0; 
FOR i:= 1 TO j DO
	rEncoderRadiansSum := rEncoderRadiansSum + rEncoderRadiansBuffer[i];
END_FOR
rEncoderRadiansFiltered := rEncoderRadiansSum / j; 


// Load cell 
fbLoadCell(); 
rGripForce := fbLoadCell.rCalibratedOutput; 


// Update globals for logging 
GVL.ENCODER_1_COUNTER_VALUE := nEncoderCounts; 
GVL.ENCODER_1_DEGREES := rEncoderDegrees;
GVL.MOTOR_1_APPLIED_VOLTAGE := rCommandVoltage; 
GVL.LOAD_CELL_NEWTONS := rGripForce;

METHOD Reset : BOOL
VAR_INPUT
END_VAR
fbEncoder1.Reset();
END_METHOD

END_FUNCTION_BLOCK

// ---- POUs/TEST.TcPOU
PROGRAM TEST
VAR
END_VAR

GVL.ENCODER_1_RAW_COUNTS;

END_PROGRAM
